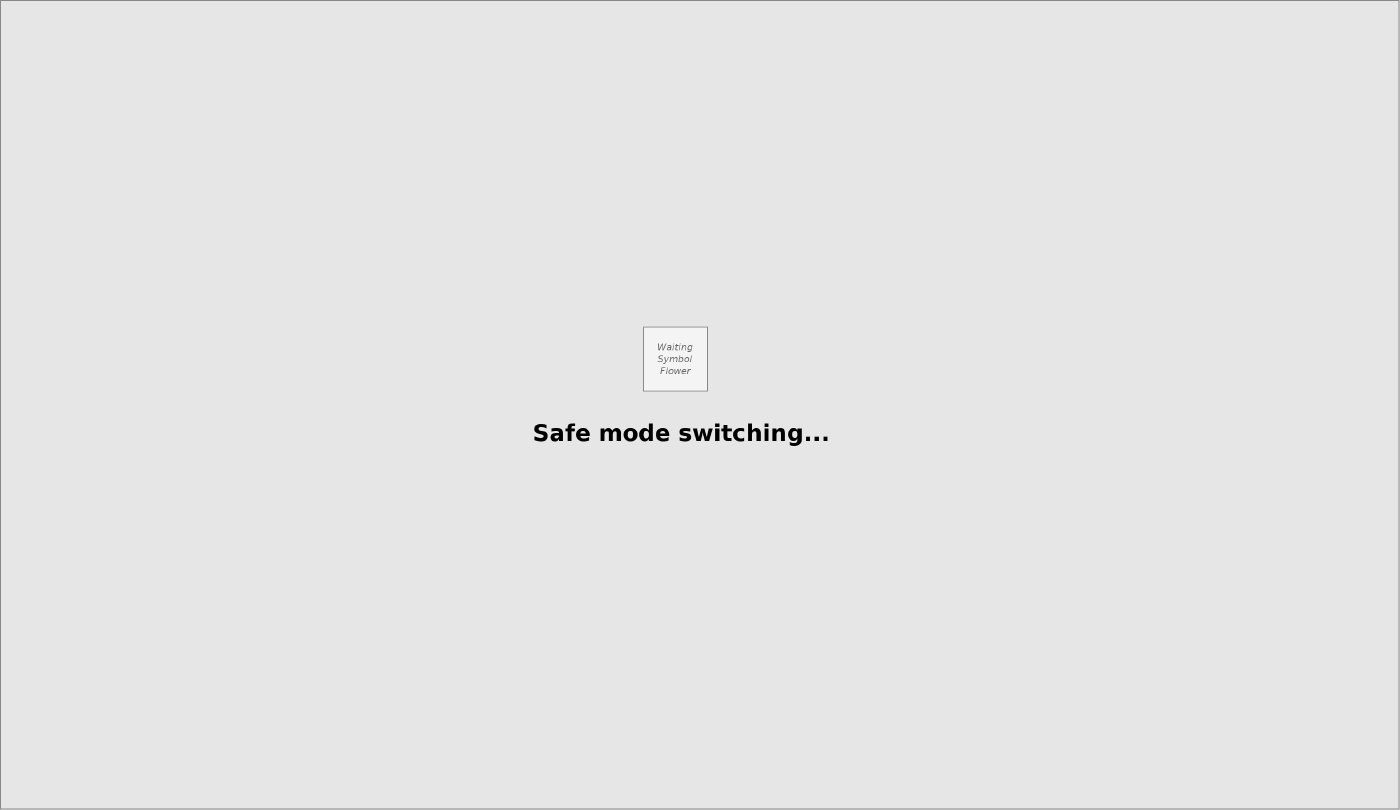
VISUALIZATION PageSwitchMode  // 1520x880
    Label (490,450 500x40), "Safe mode switching..."
    WaitingSymbolFlower (698,355 70x70)
END_VISUALIZATION

(* stored: Version 1.1.0.1, ProductVersion 3.1.4024.9
   Visu PageSwitchMode: Id {bdd43bde-a9f3-4c2d-8436-dc2f673a27f8} *)
